Omron Sysmac Studio project Colorificio (Sysmac Studio 1.30.0.17, StandardProject)
(* ù *)

# Controller PLC: NX1P2-9024DT1 version 1.40
Task PrimaryTask (priority 4, period or condition 2000): Program0
Library OmronLib_WC_Toolbox_V1_0 1.0.0 (contents left out)

TYPE S_Colori : STRUCT
    ALPHA : INT;
    RED : INT;
    GREEN : INT;
    BLU : INT;
    NOME : STRING[256];
END_STRUCT END_TYPE

VAR_GLOBAL
    SB0 : BOOL;  (* pulsante avvio ciclo automatico *)
    SB1 : BOOL;  (* pulsante arresto ciclo automatico *)
    SBE : BOOL;  (* pulsante arresto di emergenza *)
    YVA : BOOL;  (* libera caricatore seconda latta (A-) *)
    YVB : BOOL;  (* libera caricatore prima latta (B-) *)
    YVC : BOOL;  (* scarico bilancia (C+) *)
    KM1 : BOOL;  (* motore primo nastro *)
    KM2 : BOOL;  (* motore secondo nastro *)
    YVD : BOOL;  (* scarico coperchiatrice (D+) *)
    a0 : BOOL := False;  (* caricatore seconda latta libero (NA) *)
    a1 : BOOL := True;  (* caricatore seconda latta bloccato (NA) *)
    b0 : BOOL := False;  (* caricatore prima latta libero (NA) *)
    b1 : BOOL := True;  (* caricatore prima latta bloccato (NA) *)
    c0 : BOOL := True;  (* scaricatore bilancia rientrato (NA) *)
    c1 : BOOL := False;  (* scaricatore bilancia esteso (NA) *)
    d0 : BOOL := True;  (* scaricatore coperchiatrice rientrato (NA) *)
    d1 : BOOL := False;  (* scaricatore coperchiatrice esteso (NA) *)
    BIL : REAL;  (* bilancia/cella di carico (Grammi) *)
    YVBASE : BOOL;  (* eroga colorante base *)
    YVRED : BOOL;  (* eroga colorante rosso *)
    YVGREEN : BOOL;  (* eroga colorante verde *)
    YVBLU : BOOL;  (* eroga colorante blu *)
    YVSCARICO : BOOL;  (* eroga totale colore *)
    Tbase : INT;  (* tempo carico base *)
    Trosso : INT;  (* tempo carico rosso *)
    Tgreen : INT;  (* tempo carico verde *)
    Tblu : INT;  (* tempo carico blu *)
    BLW0 : BOOL := True;  (* livello minimo Base White (NA) *)
    BLW1 : BOOL := True;  (* livello riserva Base White (NA) *)
    BLR0 : BOOL := True;  (* livello minimo Red (NA) *)
    BLR1 : BOOL := True;  (* livello riserva Red (NA) *)
    BLG0 : BOOL := True;  (* livello minimo Green (NA) *)
    BLG1 : BOOL := True;  (* livello riserva Green (NA) *)
    BLB0 : BOOL := True;  (* livello minimo Blu (NA) *)
    BLB1 : BOOL := True;  (* livello riserva Blu (NA) *)
    BC0 : BOOL := False;  (* presenza prima latta sul caricatore (NA) *)
    BC1 : BOOL := False;  (* presenza seconda latta sul caricatore (NA) *)
    BBIL : BOOL := False;  (* presenza sulla bilancia (NA) *)
    BCOP : BOOL := False;  (* presenza sulla coperchiatrice (NA) *)
END_VAR

PROGRAM Program0
VAR_EXTERNAL
    SB1 : BOOL;
    KM1 : BOOL;
    YVC : BOOL;
    BBIL : BOOL;
    c0 : BOOL;
    c1 : BOOL;
    KM2 : BOOL;
    SB0 : BOOL;
    SBE : BOOL;
    BIL : REAL;
END_VAR

(* Section Section0: ladder, written here as Structured Text *)

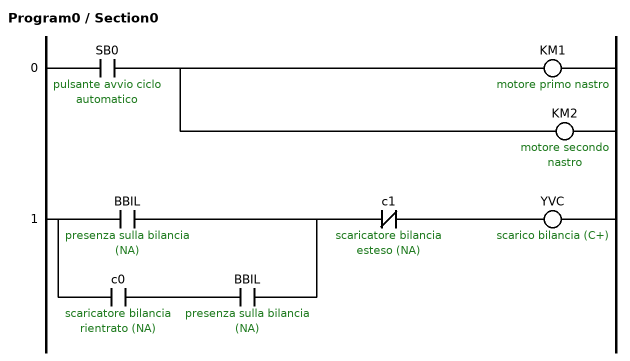
(* Rung 0 *)
KM1 := SB0;
KM2 := SB0;
(* Rung 1 *)
YVC := (BBIL OR (c0 AND BBIL)) AND NOT c1;
END_PROGRAM

FUNCTION WC_Weight : INT
VAR_INPUT
    LoadCellValue : INT;
END_VAR
// Il valore espresso è il peso in grammi
WC_Weight:=LoadCellValue*30; // LoadCellValue = livello colore della tramoggia di pesatura
END_FUNCTION

# Device HMI (NA): not converted